{attribute 'qualified_only'}
{attribute 'strict'}
TYPE E_Xelectrix_GridState_1 :
(
	eNoDataReceived := 0,
	eOff := 1,
	eIslandMode := 2,
	eOnline := 3,
	eError := 4
);
END_TYPE

(* stored: Version 1.1.0.1, ProductVersion 3.1.4024.12
   DUT E_Xelectrix_GridState_1: Id {959cbe13-f3f2-43c6-b63d-eeec03acf6ef} *)
